FUNCTION_BLOCK seek_job IMPLEMENTS InterfaceObserver
VAR_INPUT
END_VAR
VAR_OUTPUT
END_VAR
VAR
	_job_id :T_MaxString;
END_VAR

PROPERTY job_id : T_MaxString
GET
job_id := _job_id;
END_GET
SET
_job_id := job_id;
END_SET
END_PROPERTY

METHOD subscribe_job_directory : BOOL
VAR_INPUT
	(* Represent reference to subscribed job object*)
	executor	: REFERENCE TO FB_Executor;
END_VAR
END_METHOD

METHOD subscribe_job_event : BOOL
VAR_INPUT
	(* Subject text of event*)
	subject	: Tc2_System.T_MaxString;
	(* Job state before transition.*)
	old_state	: E_FutureExecutionState;
	(* Job state after transition.*)
	new_state	: E_FutureExecutionState;
	(* File-time at the time of transition.*)
	record_time	: Tc2_Utilities.T_FILETIME64;
	(* Reference to job instance of which transition occurs.*)
	executor	: REFERENCE TO FB_Executor;
END_VAR
END_METHOD

END_FUNCTION_BLOCK

(* stored: Version 1.1.0.1, ProductVersion 3.1.4024.12
   POU seek_job: Id {b598f05a-2016-4544-8790-a7d2bd225b96}, SpecialFunc None
   Property job_id: Id {05649e3c-eba0-445a-9db7-643ed3fa9cfc}
   Get Get: Id {96926441-094e-4daa-b23f-b66aa574423c}
   Set Set: Id {02620227-07c2-4cbc-b897-67a9d7a39822}
   Method subscribe_job_directory: Id {03051384-5668-4dfd-b49d-b143652b5cb3}
   Method subscribe_job_event: Id {cec237c9-50f4-4c3a-8f34-72085c243386} *)
